    stLENS1_750[842].fEnergy := 32120.253032; stLENS1_750[842].fLow := 3.813498; stLENS1_750[842].fHigh := 9.063293;
    stLENS1_750[843].fEnergy := 32184.557822; stLENS1_750[843].fLow := 3.799407; stLENS1_750[843].fHigh := 9.024741;
    stLENS1_750[844].fEnergy := 32248.991349; stLENS1_750[844].fLow := 3.785367; stLENS1_750[844].fHigh := 8.986354;
    stLENS1_750[845].fEnergy := 32313.553873; stLENS1_750[845].fLow := 3.771380; stLENS1_750[845].fHigh := 8.948129;
    stLENS1_750[846].fEnergy := 32378.245651; stLENS1_750[846].fLow := 3.757444; stLENS1_750[846].fHigh := 8.910067;
    stLENS1_750[847].fEnergy := 32443.066942; stLENS1_750[847].fLow := 3.743559; stLENS1_750[847].fHigh := 8.872167;
    stLENS1_750[848].fEnergy := 32508.018005; stLENS1_750[848].fLow := 3.729726; stLENS1_750[848].fHigh := 8.834429;
    stLENS1_750[849].fEnergy := 32573.099101; stLENS1_750[849].fLow := 3.715944; stLENS1_750[849].fHigh := 8.796851;
    stLENS1_750[850].fEnergy := 32638.310488; stLENS1_750[850].fLow := 3.702213; stLENS1_750[850].fHigh := 8.759432;
    stLENS1_750[851].fEnergy := 32703.652430; stLENS1_750[851].fLow := 3.688533; stLENS1_750[851].fHigh := 8.722173;
    stLENS1_750[852].fEnergy := 32769.125185; stLENS1_750[852].fLow := 3.674903; stLENS1_750[852].fHigh := 8.685073;
    stLENS1_750[853].fEnergy := 32834.729018; stLENS1_750[853].fLow := 3.661324; stLENS1_750[853].fHigh := 8.648130;
    stLENS1_750[854].fEnergy := 32900.464189; stLENS1_750[854].fLow := 3.647795; stLENS1_750[854].fHigh := 8.611344;
    stLENS1_750[855].fEnergy := 32966.330962; stLENS1_750[855].fLow := 3.634316; stLENS1_750[855].fHigh := 8.574715;
    stLENS1_750[856].fEnergy := 33032.329601; stLENS1_750[856].fLow := 3.620886; stLENS1_750[856].fHigh := 8.538241;
    stLENS1_750[857].fEnergy := 33098.460369; stLENS1_750[857].fLow := 3.607507; stLENS1_750[857].fHigh := 8.501923;
    stLENS1_750[858].fEnergy := 33164.723530; stLENS1_750[858].fLow := 3.594176; stLENS1_750[858].fHigh := 8.465759;
    stLENS1_750[859].fEnergy := 33231.119351; stLENS1_750[859].fLow := 3.580895; stLENS1_750[859].fHigh := 8.429749;
    stLENS1_750[860].fEnergy := 33297.648096; stLENS1_750[860].fLow := 3.567663; stLENS1_750[860].fHigh := 8.393893;
    stLENS1_750[861].fEnergy := 33364.310032; stLENS1_750[861].fLow := 3.554480; stLENS1_750[861].fHigh := 8.358188;
    stLENS1_750[862].fEnergy := 33431.105426; stLENS1_750[862].fLow := 3.541346; stLENS1_750[862].fHigh := 8.322636;
    stLENS1_750[863].fEnergy := 33498.034543; stLENS1_750[863].fLow := 3.528260; stLENS1_750[863].fHigh := 8.287235;
    stLENS1_750[864].fEnergy := 33565.097653; stLENS1_750[864].fLow := 3.515222; stLENS1_750[864].fHigh := 8.251984;
    stLENS1_750[865].fEnergy := 33632.295023; stLENS1_750[865].fLow := 3.502233; stLENS1_750[865].fHigh := 8.216883;
    stLENS1_750[866].fEnergy := 33699.626923; stLENS1_750[866].fLow := 3.489292; stLENS1_750[866].fHigh := 8.181932;
    stLENS1_750[867].fEnergy := 33767.093621; stLENS1_750[867].fLow := 3.476398; stLENS1_750[867].fHigh := 8.147129;
    stLENS1_750[868].fEnergy := 33834.695387; stLENS1_750[868].fLow := 3.463552; stLENS1_750[868].fHigh := 8.112475;
    stLENS1_750[869].fEnergy := 33902.432493; stLENS1_750[869].fLow := 3.450754; stLENS1_750[869].fHigh := 8.077968;
    stLENS1_750[870].fEnergy := 33970.305208; stLENS1_750[870].fLow := 3.438003; stLENS1_750[870].fHigh := 8.043607;
    stLENS1_750[871].fEnergy := 34038.313804; stLENS1_750[871].fLow := 3.425299; stLENS1_750[871].fHigh := 8.009393;
    stLENS1_750[872].fEnergy := 34106.458554; stLENS1_750[872].fLow := 3.412642; stLENS1_750[872].fHigh := 7.975324;
    stLENS1_750[873].fEnergy := 34174.739729; stLENS1_750[873].fLow := 3.400032; stLENS1_750[873].fHigh := 7.941400;
    stLENS1_750[874].fEnergy := 34243.157604; stLENS1_750[874].fLow := 3.387468; stLENS1_750[874].fHigh := 7.907621;
    stLENS1_750[875].fEnergy := 34311.712451; stLENS1_750[875].fLow := 3.374951; stLENS1_750[875].fHigh := 7.873985;
    stLENS1_750[876].fEnergy := 34380.404545; stLENS1_750[876].fLow := 3.362480; stLENS1_750[876].fHigh := 7.840492;
    stLENS1_750[877].fEnergy := 34449.234161; stLENS1_750[877].fLow := 3.350055; stLENS1_750[877].fHigh := 7.807142;
    stLENS1_750[878].fEnergy := 34518.201574; stLENS1_750[878].fLow := 3.337676; stLENS1_750[878].fHigh := 7.773933;
    stLENS1_750[879].fEnergy := 34587.307059; stLENS1_750[879].fLow := 3.325342; stLENS1_750[879].fHigh := 7.740866;
    stLENS1_750[880].fEnergy := 34656.550894; stLENS1_750[880].fLow := 3.313055; stLENS1_750[880].fHigh := 7.707939;
    stLENS1_750[881].fEnergy := 34725.933355; stLENS1_750[881].fLow := 3.300813; stLENS1_750[881].fHigh := 7.675153;
    stLENS1_750[882].fEnergy := 34795.454720; stLENS1_750[882].fLow := 3.288615; stLENS1_750[882].fHigh := 7.642506;
    stLENS1_750[883].fEnergy := 34865.115267; stLENS1_750[883].fLow := 3.276463; stLENS1_750[883].fHigh := 7.609998;
    stLENS1_750[884].fEnergy := 34934.915274; stLENS1_750[884].fLow := 3.264356; stLENS1_750[884].fHigh := 7.577628;
    stLENS1_750[885].fEnergy := 35004.855021; stLENS1_750[885].fLow := 3.252294; stLENS1_750[885].fHigh := 7.545396;
    stLENS1_750[886].fEnergy := 35074.934788; stLENS1_750[886].fLow := 3.240276; stLENS1_750[886].fHigh := 7.513300;
    stLENS1_750[887].fEnergy := 35145.154854; stLENS1_750[887].fLow := 3.228303; stLENS1_750[887].fHigh := 7.481342;
    stLENS1_750[888].fEnergy := 35215.515501; stLENS1_750[888].fLow := 3.216374; stLENS1_750[888].fHigh := 7.449519;
    stLENS1_750[889].fEnergy := 35286.017010; stLENS1_750[889].fLow := 3.204489; stLENS1_750[889].fHigh := 7.417832;
    stLENS1_750[890].fEnergy := 35356.659663; stLENS1_750[890].fLow := 3.192648; stLENS1_750[890].fHigh := 7.386279;
    stLENS1_750[891].fEnergy := 35427.443743; stLENS1_750[891].fLow := 3.180850; stLENS1_750[891].fHigh := 7.354861;
    stLENS1_750[892].fEnergy := 35498.369532; stLENS1_750[892].fLow := 3.169097; stLENS1_750[892].fHigh := 7.323576;
    stLENS1_750[893].fEnergy := 35569.437315; stLENS1_750[893].fLow := 3.157386; stLENS1_750[893].fHigh := 7.292425;
    stLENS1_750[894].fEnergy := 35640.647376; stLENS1_750[894].fLow := 3.145719; stLENS1_750[894].fHigh := 7.261406;
    stLENS1_750[895].fEnergy := 35712.000000; stLENS1_750[895].fLow := 3.134095; stLENS1_750[895].fHigh := 7.230519;
    stLENS1_750[896].fEnergy := 35783.495472; stLENS1_750[896].fLow := 3.122514; stLENS1_750[896].fHigh := 7.199763;
    stLENS1_750[897].fEnergy := 35855.134077; stLENS1_750[897].fLow := 3.110976; stLENS1_750[897].fHigh := 7.169138;
    stLENS1_750[898].fEnergy := 35926.916104; stLENS1_750[898].fLow := 3.099481; stLENS1_750[898].fHigh := 7.138643;

    bInitialized := TRUE;
END_IF

END_FUNCTION_BLOCK

(* stored: Version 1.1.0.1, ProductVersion 3.1.4018.10
   POU FB_EnergyTables: Id {3964a458-252f-4f9a-833e-ac7498f4c8f4}, SpecialFunc None *)
